// TIA Portal V20 export
DATA_BLOCK "SP501"   // DB317
// stored: MemoryReserve 100
   VAR
      SPARE : Bool;
      "SAFETY DC POWER TRIPPED E218CB" : Bool;
      "CLASS 2 SMPS POWER TRIPPED E308CB" : Bool;
      "CLASS 2 SMPS MONITORING E310PWS" : Bool;
      "ET200ECO PN-1 POWER TRIPPED E324CB" : Bool;
      "ET200ECO PN-2 POWER TRIPPED E328CB" : Bool;
      "ET200ECO PN-3 POWER TRIPPED E332CB" : Bool;
      "ET200ECO PN-4 POWER TRIPPED E336CB" : Bool;
      SPARE_1 : Bool;
      SPARE_2 : Bool;
      SPARE_3 : Bool;
      SPARE_4 : Bool;
      SPARE_5 : Bool;
      SPARE_6 : Bool;
      SPARE_7 : Bool;
      SPARE_8 : Bool;
   END_VAR
BEGIN
END_DATA_BLOCK
